// SIMATIC S7-200 project (STEP 7-Micro/WIN), CPU 221 REL 01.10

ORGANIZATION_BLOCK MAIN:OB1
TITLE=PROGRAM COMMENTS
BEGIN
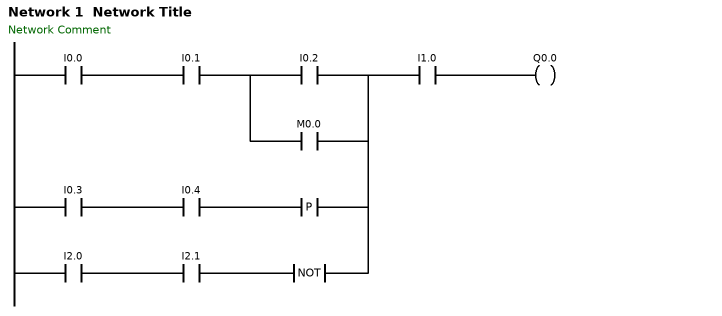
Network 1 // Network Title
// Network Comment
LD     I0.0
A      I0.1
LD     I0.2
O      M0.0
ALD
LD     I0.3
A      I0.4
EU
LD     I2.0
A      I2.1
NOT
OLD
OLD
A      I1.0
=      Q0.0
END_ORGANIZATION_BLOCK
